FUNCTION_BLOCK Fb_Counter
VAR_INPUT
END_VAR
VAR_OUTPUT
	i_countOut			: INT;
END_VAR
VAR
	i_counter_save		: INT;
	i_countUp			: INT := 1;
END_VAR

i_counter_save := i_counter_save + i_countUp;
i_countOut := i_counter_save;

END_FUNCTION_BLOCK

(* stored: Version 1.1.0.1, ProductVersion 3.1.4024.9
   POU Fb_Counter: Id {b895edcf-dd57-4356-9e4d-062f5de0beb6}, SpecialFunc None *)
